TYPE AX5000_S_0203 :
STRUCT
	Amplifier_shut_down_temperature:UINT;
END_STRUCT
END_TYPE

(* stored: Version 1.1.0.1, ProductVersion 3.1.4024.3
   DUT AX5000_S_0203: Id {9618c564-938b-44fa-ab90-7ada64a39b0e} *)
